(* IEC 61131-3 sources: Solar_and_Heat_Control/Solar_und_Heizungssteuerung/src, 5 files *)

(* ---- types.iecst ---- *)
TYPE
  Inputs : STRUCT
    ai1 : UINT;
    ai2 : UINT;
    ai3 : UINT;
    ai4 : UINT;
    ai5 : UINT;
    ai6 : UINT;
    ai7 : UINT;
    ai8 : UINT;
    ai9 : UINT;
    ai10 : UINT;
    ai11 : UINT;
    ai12 : UINT;
    ai13 : UINT;
    ai14 : UINT;
    ai15 : UINT;
    ai16 : UINT;
    ai17 : UINT;
    ai18 : UINT;
    ai19 : UINT;
    ai20 : UINT;

    di0 : BOOL;
    di1 : BOOL;
    di2 : BOOL;
    di3 : BOOL;
    di4 : BOOL;
    di5 : BOOL;
    di6 : BOOL;
    di7 : BOOL;
    di8 : BOOL;
    di9 : BOOL;
    di10 : BOOL;
    di11 : BOOL;
    di12 : BOOL;
    di13 : BOOL;
    di14 : BOOL;
    di15 : BOOL;
    di16 : BOOL;
    di17 : BOOL;
    di18 : BOOL;
    di19 : BOOL;
    di20 : BOOL;
  	di21 : BOOL;
  	di22 : BOOL;
  	di23 : BOOL;
  	Regler_R_Bit0 : BOOL;
  	Regler_L_Bit2 : BOOL;
  	Regler_R_Bit1 : BOOL;
  	Regler_L_Bit0 : BOOL;
  	Regler_L_Bit1 : BOOL;
  	Regler_R_Bit2 : BOOL;
  	di30 : BOOL;
  	di31 : BOOL;
  	active_230V : BOOL;
  	thermofuse_active : BOOL;
  	di34 : BOOL;
  	di35 : BOOL;
  	di36 : BOOL;
  	di37 : BOOL;
  	di38 : BOOL;
  	di39 : BOOL;
  END_STRUCT;
  Outputs : STRUCT
  	ao1 : UINT;
  	ao2 : UINT;
  	ao3 : UINT;
  	ao4 : UINT;

	do0 : BOOL;
  	do1 : BOOL;
  	do2 : BOOL;
  	do3 : BOOL;
  	do4 : BOOL;
  	do5 : BOOL;
  	do6 : BOOL;
  	do7 : BOOL;
  	do8 : BOOL;
  	do9 : BOOL;
  	do10 : BOOL;
  	do11 : BOOL;
  	Frostschutzventil : BOOL;
  	Solarkuehlventil : BOOL;
  	do14 : BOOL;
  	do15 : BOOL;
  	Status_LED : BOOL;
  	do17 : BOOL;
  	do18 : BOOL;
  	do19 : BOOL;
  	do20 : BOOL;
  	do21 : BOOL;
  	do22 : BOOL;
  	do23 : BOOL;
  	Pumpe4 : BOOL;
  	Pumpe3 : BOOL;
  	Pumpe2 : BOOL;
  	Pumpe1 : BOOL;
  	do28 : BOOL;
  	do29 : BOOL;
  	Wechselrichter : BOOL;
  	Spannungswandler : BOOL;
  	HK_waermer : BOOL;
  	HK_kaelter : BOOL;
  	FBH_waermer : BOOL;
  	FBH_kaelter : BOOL;
  	Schichtlader_mitte_laden : BOOL;
  	Schichtlader_fahren : BOOL;
  	Pumpe_HK : BOOL;
  	Pumpe_FBH : BOOL;
  END_STRUCT;
END_TYPE

(* ---- Prog.iecfbd ---- *)
FUNCTION_BLOCK Prog
  VAR
    R_TRIG1 : R_TRIG;
    walter : INT;
    WriteOutputs1 : WriteOutputs;
    Test : Outputs;
  END_VAR

  @VF(3) : @E(Test),@R(173.0, 197.0, 140.0, 19.0);

  (*

  *)
END_FUNCTION_BLOCK

(* ---- read_inputs.iecst ---- *)
FUNCTION_BLOCK ReadInputs
	VAR_INPUT
		inputs : REF_TO Inputs;
	END_VAR

	VAR
		data : REF_TO Inputs; /* workaround */
		fd : DINT := -1;
		analog_in_1 : ARRAY[0..4] OF UINT;
		analog_in_2 : ARRAY[0..4] OF UINT;
		analog_in_3 : ARRAY[0..4] OF UINT;
		analog_in_4 : ARRAY[0..4] OF UINT;
		digital_in_0 : ARRAY[0..7] OF BOOL;
		digital_in_1 : ARRAY[0..7] OF BOOL;
		digital_in_2 : ARRAY[0..7] OF BOOL;
		digital_in_3 : ARRAY[0..7] OF BOOL;
		digital_in_4 : ARRAY[0..7] OF BOOL;
	END_VAR

	data := inputs; /* workaround */

	/* read data from I/O sub-systems */
	IF fd < 0 THEN
		fd := I2C_Open(bus_id := 1); /* /dev/i2c-1 */
	END_IF;

	/*
	 * 0x38 ... Input 1
     * 0x39 ... Input 2
     * 0x3a ... Input 3
     * 0x3c ... Input 4
     * 0x3d ... Input 5
	 */

	IF fd >= 0 THEN
		analog_in_1 := I2HAE(fd := fd, address := 16#08);
		data^.ai6 := analog_in_1[0];
		data^.ai7 := analog_in_1[1];
		data^.ai8 := analog_in_1[2];
		data^.ai9 := analog_in_1[3];
		data^.ai10 := analog_in_1[4];

		analog_in_2 := I2HAE(fd := fd, address := 16#09);
		data^.ai1 := analog_in_2[0];
		data^.ai2 := analog_in_2[1];
		data^.ai3 := analog_in_2[2];
		data^.ai4 := analog_in_2[3];
		data^.ai5 := analog_in_2[4];

		analog_in_3 := I2HAE(fd := fd, address := 16#0A);
		data^.ai11 := analog_in_3[0];
		data^.ai12 := analog_in_3[1];
		data^.ai13 := analog_in_3[2];
		data^.ai14 := analog_in_3[3];
		data^.ai15 := analog_in_3[4];

		analog_in_4 := I2HAE(fd := fd, address := 16#0B);
		data^.ai16 := analog_in_4[0];
		data^.ai17 := analog_in_4[1];
		data^.ai18 := analog_in_4[2];
		data^.ai19 := analog_in_4[3];
		data^.ai20 := analog_in_4[4];

		digital_in_0 := I2C_PCF8574_read(fd := fd, address := 16#38);
		data^.di0 := digital_in_0[0];
		data^.di1 := digital_in_0[1];
		data^.di2 := digital_in_0[2];
		data^.di3 := digital_in_0[3];
		data^.di4 := digital_in_0[4];
		data^.di5 := digital_in_0[5];
		data^.di6 := digital_in_0[6];
		data^.di7 := digital_in_0[7];

		digital_in_1 := I2C_PCF8574_read(fd := fd, address := 16#39);
		data^.di8 := digital_in_1[0];
		data^.di9 := digital_in_1[1];
		data^.di10 := digital_in_1[2];
		data^.di11 := digital_in_1[3];
		data^.di12 := digital_in_1[4];
		data^.di13 := digital_in_1[5];
		data^.di14 := digital_in_1[6];
		data^.di15 := digital_in_1[7];

		digital_in_2 := I2C_PCF8574_read(fd := fd, address := 16#3a);
		data^.di16 := digital_in_2[0];
		data^.di17 := digital_in_2[1];
		data^.di18 := digital_in_2[2];
		data^.di19 := digital_in_2[3];
		data^.di20 := digital_in_2[4];
		data^.di21 := digital_in_2[5];
		data^.di22 := digital_in_2[6];
		data^.di23 := digital_in_2[7];

		digital_in_3 := I2C_PCF8574_read(fd := fd, address := 16#3c);
		data^.Regler_R_Bit0 := digital_in_3[0];
		data^.Regler_L_Bit2 := digital_in_3[1];
		data^.Regler_R_Bit1 := digital_in_3[2];
		data^.Regler_L_Bit0 := digital_in_3[3];
		data^.Regler_L_Bit1 := digital_in_3[4];
		data^.Regler_R_Bit2 := digital_in_3[5];
		data^.di30 := digital_in_3[6];
		data^.di31 := digital_in_3[7];

		digital_in_4 := I2C_PCF8574_read(fd := fd, address := 16#3d);
		data^.active_230V := digital_in_4[0];
		data^.thermofuse_active := digital_in_4[1];
		data^.di34 := digital_in_4[2];
		data^.di35 := digital_in_4[3];
		data^.di36 := digital_in_4[4];
		data^.di37 := digital_in_4[5];
		data^.di38 := digital_in_4[6];
		data^.di39 := digital_in_4[7];

		ENO := TRUE;
	ELSE
		ENO := FALSE; /* fd < 0 */
	END_IF;

END_FUNCTION_BLOCK

(* ---- write_outputs.iecst ---- *)
FUNCTION_BLOCK WriteOutputs
	VAR_INPUT
		outputs : REF_TO Outputs;
	END_VAR

	VAR
		fd : DINT := -1;
		cumm_do_0 : ARRAY[0..7] OF BOOL; /* cumulated digital outputs */
		cumm_do_1 : ARRAY[0..7] OF BOOL; /* cumulated digital outputs */
		cumm_do_2 : ARRAY[0..7] OF BOOL; /* cumulated digital outputs */
		cumm_do_3 : ARRAY[0..7] OF BOOL; /* cumulated digital outputs */
		cumm_do_4 : ARRAY[0..7] OF BOOL; /* cumulated digital outputs */
	END_VAR

	ENO := FALSE;

	IF fd < 0 THEN
		fd := I2C_open(bus_id := 1);
	END_IF;

	/*
	 * 0x25 ... Output 1
	 * 0x22 ... Output 2
	 * 0x20 ... Output 3
	 * 0x21 ... Output 4
	 * 0x23 ... Output 5
	 */

	IF fd >= 0 THEN
		I2HAA(fd := fd, address := 16#68, channel := 0, value := outputs^.ao1);
		I2HAA(fd := fd, address := 16#68, channel := 1, value := outputs^.ao2);
		I2HAA(fd := fd, address := 16#68, channel := 2, value := outputs^.ao3);
		I2HAA(fd := fd, address := 16#68, channel := 3, value := outputs^.ao4);

		cumm_do_0[0] := outputs^.do0;
		cumm_do_0[1] := outputs^.do1;
		cumm_do_0[2] := outputs^.do2;
		cumm_do_0[3] := outputs^.do3;
		cumm_do_0[4] := outputs^.do4;
		cumm_do_0[5] := outputs^.do5;
		cumm_do_0[6] := outputs^.do6;
		cumm_do_0[7] := outputs^.do7;
		I2C_PCF8574_write(fd := fd, address := 16#25, pin_values := cumm_do_0);

		cumm_do_1[0] := outputs^.do8;
		cumm_do_1[1] := outputs^.do9;
		cumm_do_1[2] := outputs^.do10;
		cumm_do_1[3] := outputs^.do11;
		cumm_do_1[4] := outputs^.Frostschutzventil;
		cumm_do_1[5] := outputs^.Solarkuehlventil;
		cumm_do_1[6] := outputs^.do14;
		cumm_do_1[7] := outputs^.do15;
		I2C_PCF8574_write(fd := fd, address := 16#22, pin_values := cumm_do_1);

		cumm_do_2[0] := outputs^.Status_LED;
		cumm_do_2[1] := outputs^.do17;
		cumm_do_2[2] := outputs^.do18;
		cumm_do_2[3] := outputs^.do19;
		cumm_do_2[4] := outputs^.do20;
		cumm_do_2[5] := outputs^.do21;
		cumm_do_2[6] := outputs^.do22;
		cumm_do_2[7] := outputs^.do23;
		I2C_PCF8574_write(fd := fd, address := 16#20, pin_values := cumm_do_2);

		cumm_do_3[0] := outputs^.Pumpe4;
		cumm_do_3[1] := outputs^.Pumpe3;
		cumm_do_3[2] := outputs^.Pumpe2;
		cumm_do_3[3] := outputs^.Pumpe1;
		cumm_do_3[4] := outputs^.do28;
		cumm_do_3[5] := outputs^.do29;
		cumm_do_3[6] := outputs^.Wechselrichter;
		cumm_do_3[7] := outputs^.Spannungswandler;
		I2C_PCF8574_write(fd := fd, address := 16#21, pin_values := cumm_do_3);

		cumm_do_4[0] := outputs^.HK_waermer;
		cumm_do_4[1] := outputs^.HK_kaelter;
		cumm_do_4[2] := outputs^.FBH_waermer;
		cumm_do_4[3] := outputs^.FBH_kaelter;
		cumm_do_4[4] := outputs^.Schichtlader_mitte_laden;
		cumm_do_4[5] := outputs^.Schichtlader_fahren;
		cumm_do_4[6] := outputs^.Pumpe_HK;
		cumm_do_4[7] := outputs^.Pumpe_FBH;
		I2C_PCF8574_write(fd := fd, address := 16#23, pin_values := cumm_do_4);

		ENO := TRUE;
	ELSE
		ENO := FALSE;
	END_IF;

END_FUNCTION_BLOCK

(* ---- main.iecst ---- *)
PROGRAM Heating
	VAR
		/* I/O image */
		inputs : Inputs;
		outputs : Outputs;
		HK_waermer, HK_kaelter, FBH_waermer, FBH_kaelter, WZo : BOOL;
		WR_needed_FBH_k, WR_needed_FBH_w, WR_needed_HK_w, WR_needed_HK_k,WR_needed_Schichtlader_A, WR_needed_Schichtlader_B, WR_needed:BOOL;
		i, j, k, Regler_R, Regler_L : INT;
		Dach, FBH_VL, Puffer_unten, Puffer_mitte, Puffer_oben, Waermetauscher, HK_VL, Aussen, Zimmer, FBH_Soll, HK_Soll:REAL;
		Regeltoleranz:REAL:=1; /* gibt an, wie viel Unterschied IST-SOLL bei den Heizkreisen sein darf */
		test : array[0..39] of BOOL;
		/* I/O access functions */
		read_inputs : ReadInputs;
		write_outputs : WriteOutputs;
        RTRIG_SL_A, RTRIG_SL_B : R_TRIG;
        TOF1, TOF_Reglerzyklus, TOF3, TOF4 : TOF;
        TOF_SPP1, TOF_SPP2, TOF_SPS:TOF; /* S..Solar  P...Pumpe  P...Primär/S..ekundär */
        SPP1_needed, SPP2_needed, SPS_needed :BOOL;
        SPP1_nachlaufzeit, SPP2_nachlaufzeit:TIME:=TIME#300s;
        SPS_nachlaufzeit : TIME:=TIME#30s;
        PLTD:REAL:=3; /* gibt an, ab welcher Temp-diff (Wärmetauscher-Puffer) die SPS (Solarpumpe Sekundär) laufen soll */
        Puffer_laden_sinnvoll : BOOL;
        TON_wait_4_temp_increase : TON;
        wait_for_better_efficiency,P3mustON, P3_soll_ein : BOOL;
        Schichtlader_soll_A, Schichtlader_soll_B, Schichtlader_goes_to_A : BOOL;
        TOF_SLA, TOF_SLB : TOF;
        SL_Motor_A, SL_Motor_B : BOOL;
        Schichtladeventilverfahrzeit : TIME:=TIME#30s;
        temp_increase_waiting_time : TIME:=TIME#300s;
        TON_Reglerzyklus, TON2, TON3, TON4, TON_Test, TON_Test1 : TON;
        TON_HK_waermer, TON_HK_kaelter, TON_FBH_waermer, TON_FBH_kaelter : TON;
		WR_OFF_TIME : TIME:=T#30s;
		Regler_cycle_time : TIME:=TIME#5s;
		Regler_moving_time : TIME:=TIME#1s500ms;
		alive : BOOL;
		Puffer_ratio : INT; /* Füllstand des Puffers */
		Puffer_sum : REAL; /* Puffer oben + Puffer mitte + Puffer unten */
		LED_ratio : INT;
		Status_LED : BOOL;
		LED_CYCLE_TIME : TIME:=TIME#4s;
    	LED_ON_TIME : TIME;
    	TON_LED_CYCLE : TON;
    	TOF_LED_CYCLE : TOF;
    	LED_CYCLE_REAL : REAL;
    	TOF_ratter_FBH_waermer, TOF_ratter_FBH_kaelter, TOF_ratter_HK_waermer, TOF_ratter_HK_kaelter : TOF;
		TOF_HK_Pumpennachlauf, TOF_FBH_Pumpennachlauf : TOF;
		FBH_PUMPE, HK_PUMPE : BOOL;
		TON_ERROR : TON;
		TOF_ERROR : TOF;
		Plant_ERROR : BOOL;
		Solar_Kabelbruch_ERROR : BOOL;
		Solar_Kabelkurzschluss_ERROR : BOOL;
		TOF_Spannungswandler : TOF;
		Wandler_needed : BOOL;
		TOF_WT_einfrierschutz : TOF;
		WT_needs_einfrierschutz : BOOL;
		FTRIG_loadstop : F_TRIG;
		loadstop : BOOL;
		loadstop_temp : REAL;
		TON_loadstop_reset, TON_loadstop : TON;
		TON_Ratiometer : TON;
	END_VAR

		read_inputs(inputs := REF(inputs));

	/* program logic here START */

	// Variables for default FALSE:
	WR_needed := FALSE;
	Plant_ERROR := FALSE;
	Solar_Kabelbruch_ERROR := FALSE;
	Solar_Kabelkurzschluss_ERROR :=FALSE;
	Puffer_laden_sinnvoll:=FALSE;
    SPP1_needed:=FALSE;
    SPP2_needed:=FALSE;
    wait_for_better_efficiency:=FALSE;
	P3_soll_ein:=FALSE;
    Schichtlader_soll_A:=FALSE;
    Schichtlader_soll_B:=FALSE;
	P3mustON:=FALSE;
	Schichtlader_goes_to_A:=FALSE;
    RTRIG_SL_A(CLK:=FALSE);
    outputs.Schichtlader_mitte_laden:=FALSE;
    outputs.Schichtlader_fahren:=FALSE;
	Wandler_needed := FALSE;
	WT_needs_einfrierschutz := FALSE;
	SPS_needed := FALSE;

	/* determing value for rotary switches in livingrom */
	Regler_R :=0;
	IF (inputs.Regler_R_Bit0=TRUE) THEN Regler_R := Regler_R + 1;
	END_IF;
	IF (inputs.Regler_R_Bit1=TRUE) THEN Regler_R := Regler_R + 2;
	END_IF;
	IF (inputs.Regler_R_Bit2=TRUE) THEN Regler_R := Regler_R + 4;
	END_IF;
	Regler_L :=0;
	IF (inputs.Regler_L_Bit0=TRUE) THEN Regler_L := Regler_L + 1;
    END_IF;
    IF (inputs.Regler_L_Bit1=TRUE) THEN Regler_L := Regler_L + 2;
	END_IF;
	IF (inputs.Regler_L_Bit2=TRUE) THEN Regler_L := Regler_L + 4;
	END_IF;
	IF (Regler_R=0) THEN FBH_Soll:=0;
    END_IF;
	IF (Regler_R=1) THEN FBH_Soll:=21;
    END_IF;
    IF (Regler_R=2) THEN FBH_Soll:=22;
    END_IF;
    IF (Regler_R=3) THEN FBH_Soll:=23;
    END_IF;
    IF (Regler_R=4) THEN FBH_Soll:=24;
    END_IF;
    IF (Regler_R=5) THEN FBH_Soll:=25;
    END_IF;
    IF (Regler_R=6) THEN FBH_Soll:=26;
    END_IF;
    IF (Regler_R=7) THEN FBH_Soll:=27;
    END_IF;
    IF (Regler_L=0) THEN HK_Soll:=0;
    END_IF;
    IF (Regler_L=1) THEN HK_Soll:=29;
    END_IF;
    IF (Regler_L=2) THEN HK_Soll:=35;
    END_IF;
    IF (Regler_L=3) THEN HK_Soll:=41;
    END_IF;
    IF (Regler_L=4) THEN HK_Soll:=47;
    END_IF;
    IF (Regler_L=5) THEN HK_Soll:=53;
    END_IF;
    IF (Regler_L=6) THEN HK_Soll:=59;
    END_IF;
    IF (Regler_L=7) THEN HK_Soll:=65;
    END_IF;

    /* Ist Heizung in Betrieb, so wird der Wechselrichter benötigt */
    IF Regler_L<>0 OR Regler_R<>0 THEN WR_needed:=TRUE; END_IF;

    /* Wenn Regler auf "0" steht, Heizungs-Pumpe aus */
    HK_PUMPE:=TRUE;
    IF (Regler_L=0) THEN HK_PUMPE:=FALSE; END_IF;
    TOF_HK_Pumpennachlauf(IN:=HK_PUMPE,PT:=TIME#5s);
    outputs.Pumpe_HK:=TOF_HK_Pumpennachlauf.Q;

    /* Wenn Regler auf "0" steht, Fussboden Heizungs-Pumpe aus */
    FBH_PUMPE:=TRUE;
    IF (Regler_R=0) THEN FBH_PUMPE:=FALSE; END_IF;
	TOF_FBH_Pumpennachlauf(IN:=FBH_PUMPE,PT:=TIME#5s);
    IF NOT inputs.thermofuse_active THEN outputs.Pumpe_FBH:=TOF_FBH_Pumpennachlauf.Q; END_IF;
    IF inputs.thermofuse_active THEN outputs.Pumpe_FBH:=FALSE; END_IF;

    /* Umrechnung digits zu physikalischer Größe in °C */
    Dach:=TO_REAL(inputs.ai1)*2-100;
    Waermetauscher:=TO_REAL(inputs.ai6)*0.4696-136;
    FBH_VL:=TO_REAL(inputs.ai2)*0.4696-136;
    Puffer_unten:=TO_REAL(inputs.ai3)*0.4696-136;
    Puffer_mitte:=TO_REAL(inputs.ai4)*0.4696-136;
    Puffer_oben:=TO_REAL(inputs.ai5)*0.4696-136;
    HK_VL:=TO_REAL(inputs.ai7)*0.4696-136;
    Zimmer:=TO_REAL(inputs.ai8)*0.4696-136;
    Aussen:=TO_REAL(inputs.ai9)*0.4696-136;

    /* Regelung Heizkoerperkreis */
    HK_waermer:=FALSE;
    IF (HK_VL<(HK_Soll-Regeltoleranz))THEN
    HK_waermer:=TRUE;
    END_IF;

    HK_kaelter:=FALSE;
    IF (HK_VL>(HK_Soll+Regeltoleranz))THEN
    HK_kaelter:=TRUE;
    END_IF;

    // Hier wird der Verfahr- zu Pause Rythmus bei den Heizreglern erzeugt
    TON_Reglerzyklus(IN:=NOT(TON_Reglerzyklus.Q), PT:=Regler_cycle_time);
    TOF_Reglerzyklus(IN:=TON_Reglerzyklus.Q, PT:=Regler_moving_time);

    // Stotterverhinderung: um zu verhindern, dass Output "stottert" wenn Temperaturwert gerade springt
       //Änderungsrequest muss bestimmte Zeit anstehen:
    TON_HK_waermer(IN:=HK_waermer,PT:=TIME#1s);
    TON_HK_kaelter(IN:=HK_kaelter,PT:=TIME#1s);
       // ein Änderungsrequest soll dann einen Zyklus lang anstehen
    TOF_ratter_HK_waermer(IN:=TON_HK_waermer.Q,PT:=Regler_moving_time);
    TOF_ratter_HK_kaelter(IN:=TON_HK_kaelter.Q,PT:=Regler_moving_time);
    outputs.HK_kaelter:=AND(TOF_Reglerzyklus.Q,TOF_ratter_HK_kaelter.Q);
    outputs.HK_waermer:=AND(TOF_Reglerzyklus.Q,TOF_ratter_HK_waermer.Q);

    /* Regelung Fussbodenheizungskreis */
    FBH_waermer:=FALSE;
    IF (FBH_VL<(FBH_Soll-Regeltoleranz))THEN
    FBH_waermer:=TRUE;
    END_IF;

    FBH_kaelter:=FALSE;
    IF (FBH_VL>(FBH_Soll+Regeltoleranz))THEN
    FBH_kaelter:=TRUE;
    END_IF;

    // Stotterverhinderung: um zu verhindern, dass Output "stottert" wenn Temperaturwert gerade springt"
       //Änderungsrequest muss bestimmte Zeit anstehen:
    TON_FBH_waermer(IN:=FBH_waermer,PT:=TIME#1s);
    TON_FBH_kaelter(IN:=FBH_kaelter,PT:=TIME#1s);
       // ein Änderungsrequest soll dann einen Zyklus lang anstehen
    TOF_ratter_FBH_waermer(IN:=TON_FBH_waermer.Q,PT:=Regler_moving_time);
    TOF_ratter_FBH_kaelter(IN:=TON_FBH_kaelter.Q,PT:=Regler_moving_time);
    outputs.FBH_kaelter:=AND(TOF_Reglerzyklus.Q,TOF_ratter_FBH_kaelter.Q);
    outputs.FBH_waermer:=AND(TOF_Reglerzyklus.Q,TOF_ratter_FBH_waermer.Q);

    // Anlagenfehlerfaelle
    IF inputs.thermofuse_active THEN Plant_ERROR:=TRUE; END_IF;
    IF outputs.Wechselrichter AND NOT(inputs.active_230V) THEN Plant_ERROR:=TRUE; END_IF;
    IF inputs.ai1>750 OR inputs.ai6>750 OR inputs.ai3>750 OR inputs.ai4>750 OR inputs.ai5>750 THEN Solar_Kabelbruch_ERROR:=TRUE; END_IF;
    IF inputs.ai1<10 OR inputs.ai6<10 OR inputs.ai3<10 OR inputs.ai4<10 OR inputs.ai5<10 THEN Solar_Kabelkurzschluss_ERROR:=TRUE; END_IF;
    IF Solar_Kabelbruch_ERROR OR Solar_Kabelkurzschluss_ERROR THEN Plant_ERROR:=TRUE; END_IF;

    // Status - LED
    TON_LED_CYCLE(IN:=NOT(TON_LED_CYCLE.Q),PT:=LED_CYCLE_TIME);
    LED_CYCLE_REAL:=TO_REAL(IN:=LED_CYCLE_TIME);
    LED_CYCLE_REAL:=LED_CYCLE_REAL/100*Puffer_ratio;
    LED_ON_TIME:=TO_TIME(IN:=LED_CYCLE_REAL);
    TOF_LED_CYCLE(IN:=TON_LED_CYCLE.Q,PT:=LED_ON_TIME);
    TON_ERROR(IN:=NOT(TON_ERROR.Q),PT:=TIME#1s);
    TOF_ERROR(IN:=TON_ERROR.Q,PT:=TIME#500ms);
    IF NOT(Plant_ERROR) THEN outputs.status_led:=TOF_LED_CYCLE.Q;
    ELSE outputs.status_led:=TOF_ERROR.Q; END_IF;

    /* SOLAR - STEUERUNG */

	/* Einschalten der ersten Pumpe bei 35° und Dachtemp > Puffer-mitte */
    IF(Dach>(Puffer_unten+10)) THEN
      SPP1_needed:=TRUE;
      WR_needed:=TRUE;
      outputs.Frostschutzventil:=TRUE;
    END_IF;

    // outputs.Solarkuehlventil:=FALSE;

    // Übergangslösung:
    IF Dach<29 THEN outputs.Frostschutzventil:=FALSE; END_IF;

    /* Einschalten der zweiten Pumpe bei 50° */
    IF(Dach>50) THEN
      SPP2_needed:=TRUE;
    END_IF;

    /* Ist die Temp für oben noch zu klein, warten... */
    IF(Waermetauscher<Puffer_oben) AND Dach>(Puffer_unten+5) THEN
		wait_for_better_efficiency:=TRUE;
	END_IF;
    TON_wait_4_temp_increase(IN:=wait_for_better_efficiency, PT:=temp_increase_waiting_time);

    /* Waermetauschertemperatur höher als Puffer oben, muss P3 laufen. Schichtladerstellung_A sinnvoll */
    IF ((Waermetauscher-PLTD)>Puffer_oben) THEN
    	SPS_needed:=TRUE;
    	Schichtlader_soll_A:=TRUE;
    	WR_needed:=TRUE;
    END_IF;

    /* Solaranlage heizt, aber nicht genug für oben,...   ... dann unten (unten, nicht mitte!)! */
    IF(Waermetauscher-PLTD)>Puffer_unten AND TON_wait_4_temp_increase.Q THEN
    	SPS_needed:=TRUE;
    	Schichtlader_soll_B:=TRUE;
    	WR_needed:=TRUE;
    END_IF;

    // Anfahren der A-Stellung = Puffer oben laden
    IF Schichtlader_soll_A THEN
    	outputs.Schichtlader_fahren:=TRUE;
    END_IF;

	// Anfahren der B-Stellung = Puffer mittig laden
    IF Schichtlader_soll_B THEN
    	outputs.Schichtlader_mitte_laden:=TRUE;
    	outputs.Schichtlader_fahren:=TRUE;
    END_IF;

    /* Ansteuerung der Pumpen mit Nachlaufzeit */
    TOF_SPP1(IN:=SPP1_needed,PT:=SPP1_nachlaufzeit);
    TOF_SPP2(IN:=SPP2_needed,PT:=SPP2_nachlaufzeit);
    TOF_SPS(IN:=SPS_needed,PT:=SPS_nachlaufzeit);
    outputs.pumpe1:=TOF_SPP1.Q;
    outputs.pumpe2:=TOF_SPP2.Q;
    outputs.pumpe3:=TOF_SPS.Q;

    //Pufferladung (SPS) stoppt

    // Pufferladung stoppt, Primärpumpen aus
    FTRIG_loadstop(CLK:=outputs.pumpe3);
    IF FTRIG_loadstop.Q THEN loadstop:=TRUE; loadstop_temp:=Dach; END_IF;
    TON_loadstop_reset(IN:=loadstop,PT:=TIME#4h);
    IF TON_loadstop_reset.Q THEN loadstop:=FALSE; END_IF;
    IF loadstop AND (Dach+PLTD) > loadstop_temp THEN loadstop:=FALSE; END_IF;
    TON_loadstop(IN:=loadstop,PT:=TIME#5m);
    IF TON_loadstop.Q THEN outputs.pumpe1:=FALSE; outputs.pumpe2:=FALSE; END_IF;

    /* Spannungswandler ausschalten, wenn nicht mehr gebraucht */
    IF SPP1_needed OR SPP2_needed OR SPS_needed THEN Wandler_needed:=TRUE; END_IF;
    TOF_Spannungswandler(IN:=Wandler_needed,PT:=TIME#1m);
    outputs.Spannungswandler:=TOF_Spannungswandler.Q;

    // Einfrierschutz und Pumpenübertemperaturschutz
    IF Dach<4 OR Dach>120 THEN
    	outputs.pumpe1:=FALSE;
    	outputs.pumpe2:=FALSE;
    	outputs.pumpe3:=FALSE;
    END_IF;

    // Falls Ventil versagt, soll vor dem Einfrieren mit Heizwasser gewärmt werden
    IF Waermetauscher<4 THEN WT_needs_einfrierschutz:=TRUE; Wandler_needed:=TRUE; Plant_Error:=TRUE; END_IF;
    TOF_WT_einfrierschutz(IN:=WT_needs_einfrierschutz,PT:=TIME#5m);
	IF Waermetauscher<6 THEN outputs.pumpe3:=TOF_WT_einfrierschutz.Q; END_IF;

    /* Füllstand des Puffers (in %) berechnen alles: 25°C=leer, alles: 75°C ist voll*/
    Puffer_sum:=Puffer_oben + Puffer_mitte + Puffer_unten;
    Puffer_sum:=((Puffer_sum / 3) - 25) * 2;
    Puffer_ratio:=TO_INT(Puffer_sum);
    TON_Ratiometer(IN:=NOT(TON_Ratiometer.Q),PT:=TIME#1m);
    IF Puffer_ratio>0 AND TON_Ratiometer.Q THEN outputs.ao1:=TO_UINT(Puffer_ratio*9); END_IF;
    IF Puffer_ratio<=0 AND TON_Ratiometer.Q THEN outputs.ao1:=0;
    END_IF;

    /* Wechselrichter schaltet ausschaltverzögert aus */
    TOF1(PT:=WR_OFF_TIME,IN:=WR_needed);
    outputs.Wechselrichter:=TOF1.Q;

    /* program logic here END */
	write_outputs(outputs := REF(outputs));

END_PROGRAM
// LAST CHANGES
//
// 31. 1. AO1 Berechnung konnte negativ werden, wait4betterefficiency war Dachtempunabh!!!
// 31. 1. Mischer warm und kalt gleichzeitig fahren unterbunden, UINT statt USINT beim ao1, SPPs aus bei längerem nicht gebrauch
//
/* WICHTIGES:
 * Wie viele Schreibzylen/SPS Programmupdates schätzt RPo ein, dass möglich sind.
 */
